{attribute 'GeneratedUsingTerminal: EL3681-0000-0017'}
{attribute addProperty BoxType "EL3681-0000-0017"}
{attribute addProperty Id "EtcSlaveTerminalBaseSAI_InputsAT %I*SAI_Inputs_3A838E1114SAI_RangeAT %I*SAI_Range_C3200E782SAI_Range_1AT %Q*SAI_Range_3710D7473WcStateAT %I*WcState_9091E0EB2InfoDataAT %I*InfoData_32EB74EA10"}
{attribute addProperty CRC "2560085704"}
{attribute addProperty Size "31"}
TYPE EL3681_9897CEC8 EXTENDS EtcSlaveTerminalBase :
STRUCT
	{attribute addProperty Name "SAI_Inputs"}
	SAI_Inputs : SAI_Inputs_3A838E11;
	{attribute addProperty Name "SAI_Range"}
	SAI_Range : SAI_Range_C3200E78;
	{attribute addProperty Name "SAI_Range_1"}
	SAI_Range_1 : SAI_Range_3710D747;
	{attribute addProperty Name "WcState"}
	WcState : WcState_9091E0EB;
	{attribute addProperty Name "InfoData"}
	InfoData : InfoData_32EB74EA;
END_STRUCT
END_TYPE

(* stored: Version 1.2.0.0, ProductVersion 3.1.4024.9
   DUT EL3681_9897CEC8: Id {6ef5ef33-0ba2-44b7-bc31-568037b2d83e} *)
